FUNCTION_BLOCK POU EXTENDS FB_Axis
VAR_INPUT
END_VAR
VAR_OUTPUT
END_VAR
VAR
END_VAR

END_FUNCTION_BLOCK

(* stored: Version 1.1.0.1, ProductVersion 3.1.4024.11
   POU POU: Id {f86a71e7-b6ec-436c-bbc1-43616b1ea00b}, SpecialFunc None *)
